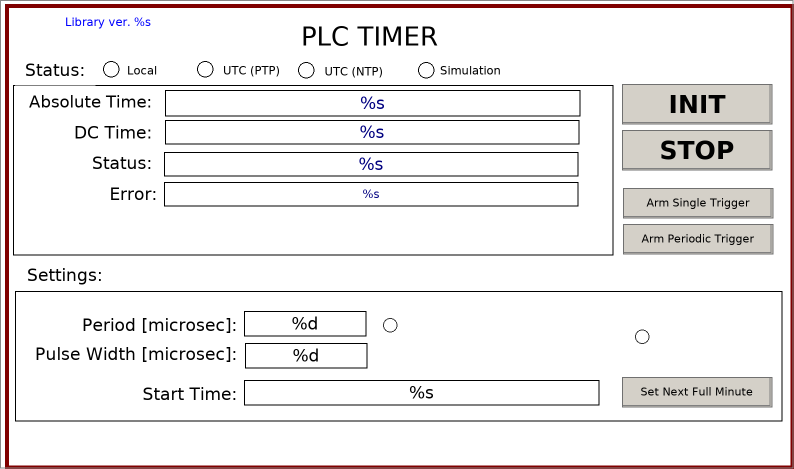
VISUALIZATION GUI_TEMPLATE_TIMER  // 794x469
VAR_IN_OUT
	m_Instance:	FB_TIMER;
END_VAR
    RoundedRectangle (5,4 789x465)
    Rectangle (13,85 600x170)
    Rectangle (15,291 767x130)
    Rectangle (15,260 100x30), "Settings:"
    Rectangle (40,315 200x20), "Period [microsec]:"
    Rectangle (30,90 125x24), "Absolute Time:"
    RoundedRectangle (245,19 249x35), "PLC TIMER"
    Rectangle (40,384 200x20), "Start Time:"
    Rectangle (165,90 415x26), "%s", text variable: m_Instance.fbTimerRef.stat.sUtcTime
    Rectangle (15,55 80x30), "Status:"
    Rectangle (244,380 355x25), "%s", text variable: m_Instance.ctrl.sStartTime
        OnMouseDown: write the text variable via Edit
    Rectangle (244,311 122x25), "%d", tooltip "Min 10 microsec", text variable: m_Instance.ctrl.nPeriod
        OnMouseDown: write the text variable via Edit, min 10
    Rectangle (35,153 120x20), "Status:"
    Rectangle (35,120 120x25), "DC Time:"
    Rectangle (165,120 414x24), "%s", text variable: m_Instance.fbTimerRef.stat.sDcTime
    Button (622,377 150x30), "Set Next Full Minute"
        OnMouseDown: execute { m_Instance.ctrl.nCommand := E_TIMER_COMMAND.COMMAND_TIMER_NEXT_MINUTE; m_Instance.ctrl.bExecute := true; }
    Button (623,188 150x30), "Arm Single Trigger"
        OnMouseDown: execute {
            m_Instance.ctrl.nCommand := E_TIMER_COMMAND.COMMAND_TIMER_ARM;
            m_Instance.ctrl.bPeriodic := FALSE;
            m_Instance.ctrl.bExecute := TRUE;
        }
    Button (622,130 150x40), "STOP"
        OnMouseDown: execute { m_Instance.ctrl.nCommand := E_TIMER_COMMAND.COMMAND_TIMER_STOP; m_Instance.ctrl.bExecute := TRUE; }
    Button (623,224 150x30), "Arm Periodic Trigger"
        OnMouseDown: execute {
            m_Instance.ctrl.nCommand := E_TIMER_COMMAND.COMMAND_TIMER_ARM;
            m_Instance.ctrl.bPeriodic := TRUE;
            m_Instance.ctrl.bExecute := TRUE;
        }
    RadioButton (381,312 103x26), variable: not m_Instance.stat.bPeriodic
        Areas[0]: Text=Periodic
    Rectangle (40,344 200x20), "Pulse Width [microsec]:"
    Rectangle (245,343 122x25), "%d", tooltip "Range 5..1000 microsec", text variable: m_Instance.ctrl.nPulseWidth
        OnMouseDown: write the text variable via Edit, min 5, max 1000
    RadioButton (633,298 118x77), variable: m_Instance.ctrl.nChannel, input disabled if: false
        Areas[0]: Text=Ch1
        Areas[1]: Text=Ch2
        Areas[2]: Text=Ch1 + Ch2
    Button (622,84 150x40), "INIT"
        OnMouseDown: execute { m_Instance.ctrl.nCommand := E_TIMER_COMMAND.COMMAND_TIMER_INIT; m_Instance.ctrl.bExecute := TRUE; }
    Rectangle (164,152 414x24), "%s", text variable: m_Instance.stat.sStatus, input disabled if: true
    Rectangle (164,182 414x24), "%s", text variable: m_Instance.stat.sErrorText, input disabled if: true
    Rectangle (40,184 120x20), "Error:", input disabled if: true
    Rectangle (62,12 145x20), "Library ver. %s", text variable: m_Instance.stat.sLibVersion
    Ellipse (103,61 16x16), tooltip "Active time: Local", colour toggle: (m_Instance.fbTimerRef.stat.mode) = E_TIME_MODE.LOCAL
    Label (116,58 44x25), "Local"
    Ellipse (197,61 16x16), tooltip "Active time: UTC", colour toggle: (m_Instance.fbTimerRef.stat.mode = E_TIME_MODE.UTC_PTP)
    Ellipse (418,62 16x16), tooltip "Active time: Simulated", colour toggle: (m_Instance.fbTimerRef.stat.mode) = E_TIME_MODE.SIMULATION
    Label (436,58 68x25), "Simulation"
    Label (212,58 71x25), "UTC (PTP)"
    Label (316,59 70x25), "UTC (NTP)"
    Ellipse (298,62 16x16), tooltip "Active time: UTC", colour toggle: (m_Instance.fbTimerRef.stat.mode = E_TIME_MODE.UTC_NTP)
END_VISUALIZATION

(* stored: Version 1.1.0.1, ProductVersion 3.1.4024.11
   Visu GUI_TEMPLATE_TIMER: Id {3ead127f-6803-4292-b24f-7196919e589b} *)
